FUNCTION_BLOCK TriggerNot0 (* Basic Function Block Type *)
  (* Standard: 61499-2 *)
  (* Version 0.0, 6/11/2026, Schneider Electric, Template *)
  PACKAGE SE.Nereda;
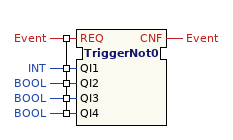
  EVENT_INPUT
    REQ WITH QI1, QI2, QI3, QI4; (* Normal Execution Request *)
  END_EVENT
  EVENT_OUTPUT
    CNF; (* Execution Confirmation *)
  END_EVENT
  VAR_INPUT
    QI1 : INT; (* Input event qualifier *)
    QI2 : BOOL;
    QI3 : BOOL;
    QI4 : BOOL;
  END_VAR
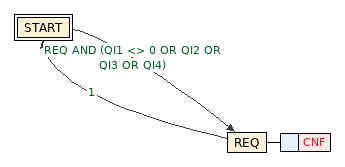
  EC_STATES
    START; (* Initial State *)
    REQ : -> CNF; (* Normal execution *)
  END_STATES
  EC_TRANSITIONS
    START TO REQ := REQ AND (QI1 <> 0 OR QI2 OR QI3 OR QI4);
    REQ TO START := 1;
  END_TRANSITIONS
END_FUNCTION_BLOCK
